{attribute 'GeneratedUsingTerminal: EL6201-0000-0017'}
{attribute addProperty BoxType "EL6201-0000-0017"}
{attribute addProperty Id "Slave_30A_DO0BOOL1Slave_30A_DO1BOOL1Slave_30A_DO2BOOL1Slave_30A_DO3BOOL1Slave_30B_DO0BOOL1Slave_30B_DO1BOOL1Slave_30B_DO2BOOL1Slave_30B_DO3BOOL1"}
{attribute addProperty CRC "395618333"}
{attribute addProperty Size "8"}
TYPE Slave_30_Outputs_1794A81D :
STRUCT
	{attribute addProperty Name "Slave_30A_DO0"}
	Slave_30A_DO0 : BOOL;
	{attribute addProperty Name "Slave_30A_DO1"}
	Slave_30A_DO1 : BOOL;
	{attribute addProperty Name "Slave_30A_DO2"}
	Slave_30A_DO2 : BOOL;
	{attribute addProperty Name "Slave_30A_DO3"}
	Slave_30A_DO3 : BOOL;
	{attribute addProperty Name "Slave_30B_DO0"}
	Slave_30B_DO0 : BOOL;
	{attribute addProperty Name "Slave_30B_DO1"}
	Slave_30B_DO1 : BOOL;
	{attribute addProperty Name "Slave_30B_DO2"}
	Slave_30B_DO2 : BOOL;
	{attribute addProperty Name "Slave_30B_DO3"}
	Slave_30B_DO3 : BOOL;
END_STRUCT
END_TYPE

(* stored: Version 1.2.0.0, ProductVersion 3.1.4024.9
   DUT Slave_30_Outputs_1794A81D: Id {fd5c8ed8-344e-4176-88ba-a869285c915c} *)
